# EPICS substitutions: qeVCLTestApp/Db/dbl_slit_test.substitutions
# File: qeVCLTestApp/Db/dbl_slit_test.substitutions
# DateTime: Mon May 26 17:17:29 2025
# Last checked in by: starritt
#

file db/dbl_slit_test.template {
    pattern { DEVICE                      }
            { "SR12ID01SLT21:HCENTRE_VRT" }
            { "SR12ID01SLT21:HSIZE_VRT"   }
            { "SR12ID01SLT21:VCENTRE_VRT" }
            { "SR12ID01SLT21:VSIZE_VRT"   }
            { "SR12ID01SLT21:XI_MTR"      }
            { "SR12ID01SLT21:XO_MTR"      }
            { "SR12ID01SLT21:YB_MTR"      }
            { "SR12ID01SLT21:YT_MTR"      }
}

# end
